PROGRAM main
  VAR
    Machine_Start_Timer : TON;
    Start_Button AT %IX0.0 : BOOL;
    Stop_Button AT %IX0.1 : BOOL;
    Emergency_Stop_Button AT %IX0.3 : BOOL;
    LED AT %QX0.0 : BOOL;
    Motor_1 AT %QX0.1 : BOOL;
    Motor_2 AT %QX0.2 : BOOL;
    Linear_actuator AT %QX0.3 : BOOL;
    Filling_Process AT %QX0.4 : BOOL;
    P_Sensor AT %IX0.4 : BOOL;
    C_Sensor AT %IX0.5 : BOOL;
    Half_Filled AT %IX0.6 : BOOL;
    TP0 : TP;
    TP1 : TP;
    TP2 : TP;
    Semi_Filled AT %QX0.5 : BOOL;
  END_VAR

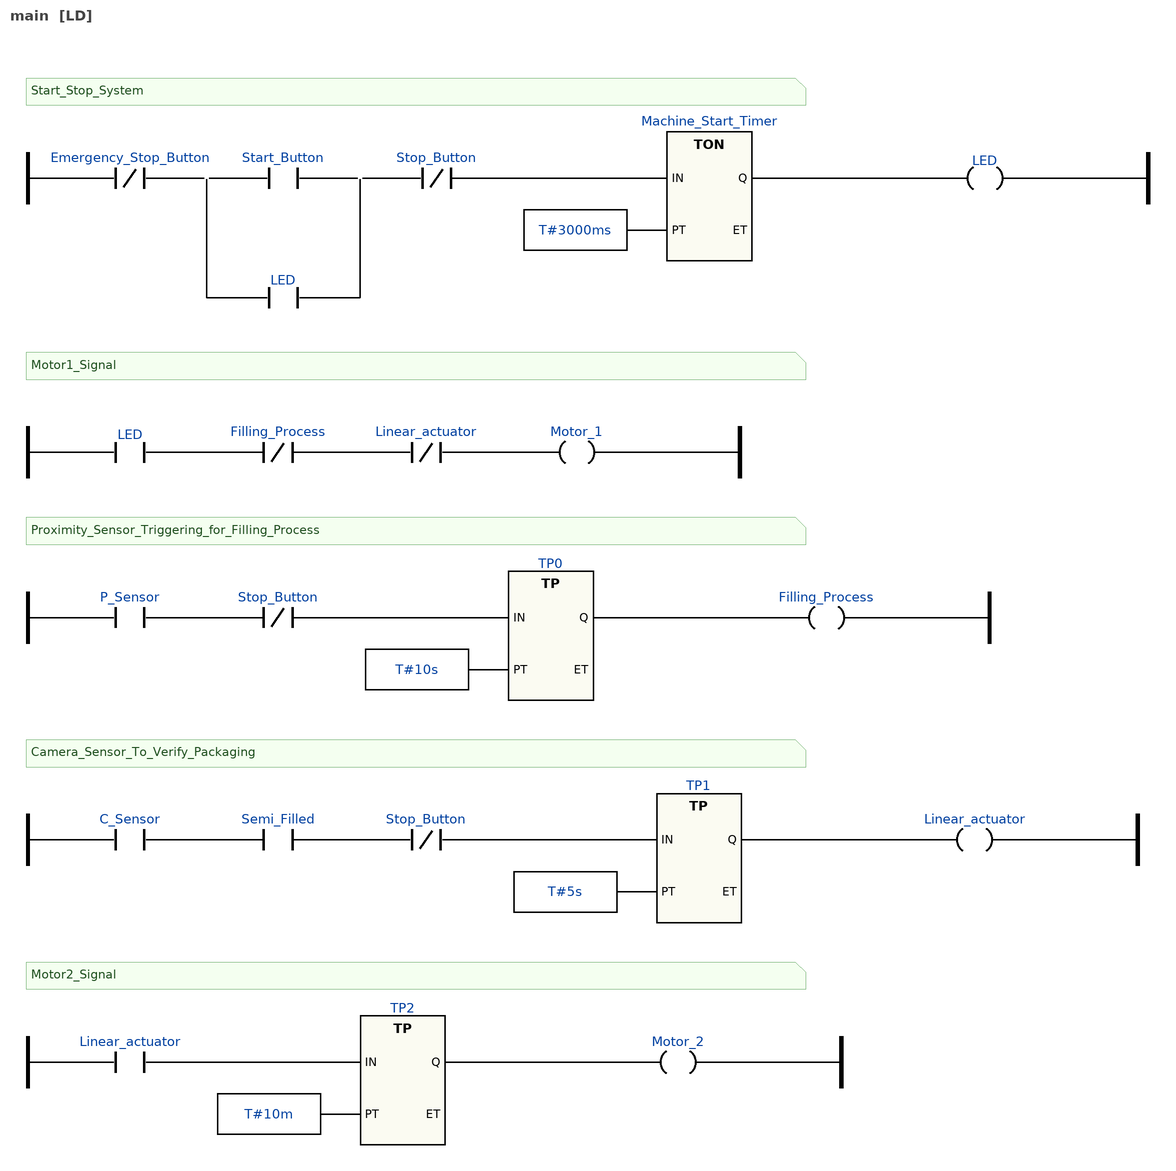
(* LD diagram, written out as Structured Text *)
(* Start_Stop_System *)
Machine_Start_Timer(IN := NOT Emergency_Stop_Button AND (Start_Button OR LED) AND NOT Stop_Button, PT := T#3000ms);
LED := Machine_Start_Timer.Q;
(* Motor1_Signal *)
Motor_1 := LED AND NOT Filling_Process AND NOT Linear_actuator;
(* Proximity_Sensor_Triggering_for_Filling_Process *)
TP0(IN := P_Sensor AND NOT Stop_Button, PT := T#10s);
Filling_Process := TP0.Q;
(* Camera_Sensor_To_Verify_Packaging *)
TP1(IN := C_Sensor AND Semi_Filled AND NOT Stop_Button, PT := T#5s);
Linear_actuator := TP1.Q;
(* Motor2_Signal *)
TP2(IN := Linear_actuator, PT := T#10m);
Motor_2 := TP2.Q;
END_PROGRAM
